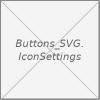
VISUALIZATION ButtonSettings  // 100x100
VAR_IN_OUT
	bState : BOOL;
END_VAR
    Frame (0,0 100x100)
        shows ButtonTemplate(bActive := bState)
    Image (0,0 100x100), image: Buttons_SVG.IconSettings
        OnMouseDown: execute { GVL_HMI.fbHMIControl.eScreenRequest := E_BaseVisu.Settings; }
END_VISUALIZATION

(* stored: Version 1.1.0.1, ProductVersion 3.1.4024.11
   Visu ButtonSettings: Id {54874a1c-cc00-424b-9eab-49a86a13f0cd} *)
